FUNCTION_BLOCK "G310M_Code"
TITLE =G310M PLC1 TO EXCISTING DEGERMINATION SYSTEM
//COPYRIGHT:    (C) 2009  BUHLER AG, CH-9240 UZWIL, SWITZERLAND
//
//PRODUCT:      WinCoS_BIW01_09
//
//TITLE:        PLC1 TO EXCISTING DEGERMINATION SYSTEM
//                Machine group control
//                Maschinengruppensteuerung
//
//--------------------------------------------------------------------------------
//
//IDENT:        AUTHOR:             DEPT:                              DATE:
//
//P01_FB410.1.0 K.Renz              CSB41                              28.Jun.2010
//             1st Release
//
//--------------------------------------------------------------------------------
//
//PURPOSE:
//
//MANUAL :
//
//RESTRICTIONS:
//
//--------------------------------------------------------------------------------
AUTHOR : KR
FAMILY : USW
VERSION : 9.9


VAR
  Gr : "GCS7_GrpCtrlSub";	//Standard interface to group
  InOutValue1 : DINT ;	//Data for user
  InOutValue2 : DINT ;	//Data for user
  OutWayConflict : BOOL ;	//Data for user
  OutSelectionOk : BOOL ;	//Data for user
  CmdNewValue : BOOL ;	//Data for user
  CmdNewJob : BOOL ;	//Data for user
  OutCodeOK : BOOL ;	//Data for user
  InEndOfJob : BOOL ;	//Data for user
  staWayOk : BOOL ;	//Data for user
  EdgeStartRelease : BOOL ;	//Data for user
  USW8 : BOOL ;	//Data for user
  USW9 : BOOL ;	//Data for user
  USW10 : BOOL ;	//Data for user
  USW11 : BOOL ;	//Data for user
  USW12 : BOOL ;	//Data for user
  USW13 : BOOL ;	//Data for user
  USW14 : BOOL ;	//Data for user
  USW15 : BOOL ;	//Data for user
  A_3956_KCL01 : "GCS7_E_DigInput";	// DigInpCont
END_VAR
VAR_TEMP
  tmpEnable : BOOL ;
  tmpFlag : BOOL ;
  tmpCmdNext : BOOL ;
  tmpLocal : BOOL ;
  tmpAspOk : BOOL ;
  tmpHWStop : BOOL ;
  tmpInstanzDBNo : INT ;
END_VAR
BEGIN
NETWORK
TITLE =



NETWORK
TITLE =Read command from group control
//Parameter
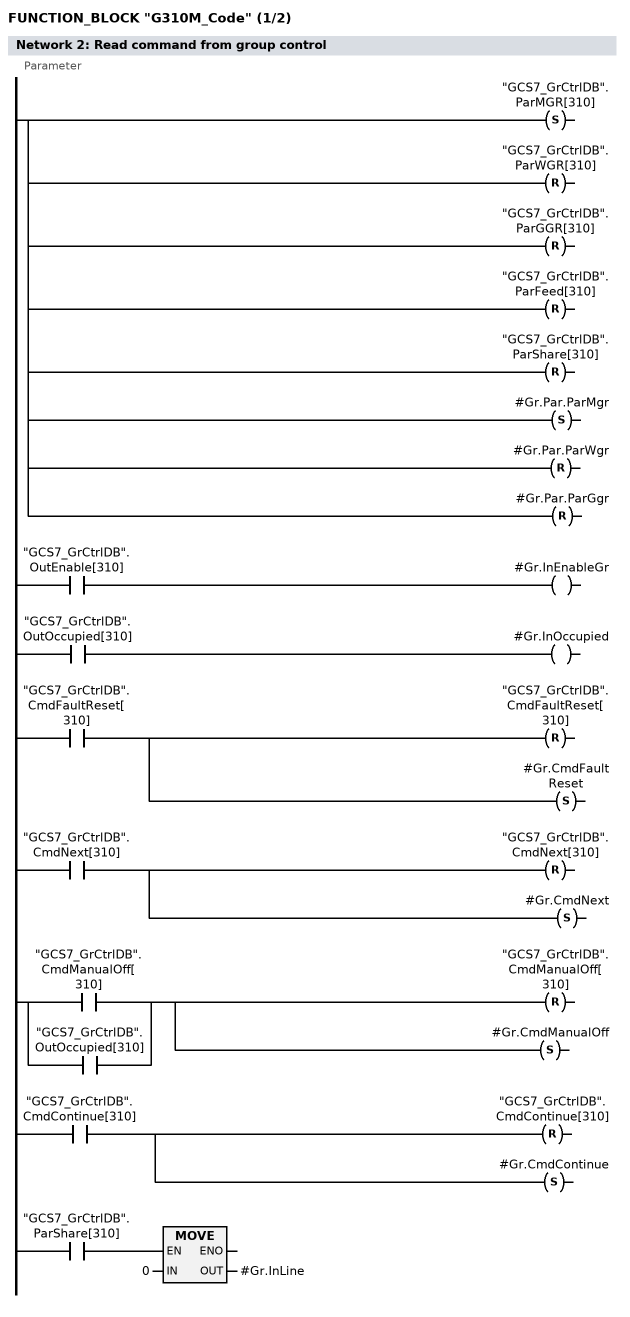
      SET   ;
      S     "GCS7_GrCtrlDB".ParMGR[310];
      R     "GCS7_GrCtrlDB".ParWGR[310];
      R     "GCS7_GrCtrlDB".ParGGR[310];
      R     "GCS7_GrCtrlDB".ParFeed[310];
      R     "GCS7_GrCtrlDB".ParShare[310];
      S     #Gr.Par.ParMgr;
      R     #Gr.Par.ParWgr;
      R     #Gr.Par.ParGgr;
//Command
      U     "GCS7_GrCtrlDB".OutEnable[310];
      =     #Gr.InEnableGr;
      U     "GCS7_GrCtrlDB".OutOccupied[310];
      =     #Gr.InOccupied;
      U     "GCS7_GrCtrlDB".CmdFaultReset[310];
      R     "GCS7_GrCtrlDB".CmdFaultReset[310];
      S     #Gr.CmdFaultReset;
      U     "GCS7_GrCtrlDB".CmdNext[310];
      R     "GCS7_GrCtrlDB".CmdNext[310];
      S     #Gr.CmdNext;
      U     "GCS7_GrCtrlDB".CmdManualOff[310];
      O     "GCS7_GrCtrlDB".OutOccupied[310];
      R     "GCS7_GrCtrlDB".CmdManualOff[310];
      S     #Gr.CmdManualOff;
      U     "GCS7_GrCtrlDB".CmdContinue[310];
      R     "GCS7_GrCtrlDB".CmdContinue[310];
      S     #Gr.CmdContinue;
//Init Line Number
      U     "GCS7_GrCtrlDB".ParShare[310];
      SPBN  WE00;
      L     0;
      T     #Gr.InLine;
WE00: NOP   0;
NETWORK
TITLE =Call Methode Control
// 1. Handle Interface PCControl
// 2. Prepare mode --> ModePassive,ModeActive,ModeIdling
// 3. Reset global flags of the group
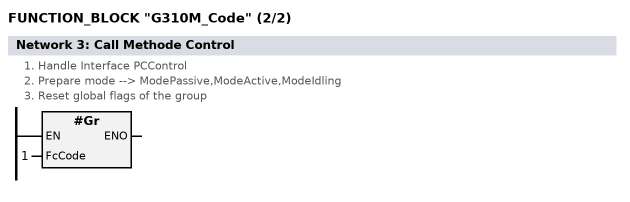
      CALL #Gr (
           FcCode                   := 1);
NETWORK
TITLE =Restart Idling Time

      L     #Gr.Par.ParIdling;
      L     2;
      >=I   ;
      SPB   IdTm;
      T     #Gr.Par.ParIdling;
IdTm: NOP   0;
      CLR   ;
      S     #Gr.CmdRestartIdling;
NETWORK
TITLE =Prepare global flags



NETWORK
TITLE =Set Pattern (Target position)



NETWORK
TITLE =Interlocking WayOk



NETWORK
TITLE =Interlocking Autostart

      CLR   ;
      R     #Gr.OutAutostart;
NETWORK
TITLE =Interlocking Enable
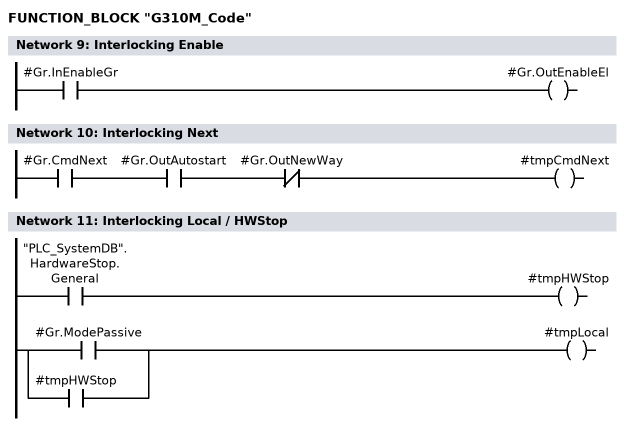

      U     #Gr.InEnableGr;
      =     #Gr.OutEnableEl;

NETWORK
TITLE =Interlocking Next

      U     #Gr.CmdNext;
      U     #Gr.OutAutostart;
      UN    #Gr.OutNewWay;
      =     #tmpCmdNext;

NETWORK
TITLE =Interlocking Local / HWStop

      U     "PLC_SystemDB".HardwareStop.General;
      =     #tmpHWStop;

      U     #Gr.ModePassive;
      O     #tmpHWStop;
      =     #tmpLocal;

NETWORK
TITLE =Interlocking Start Warning

      NOP   0;
//- Restart after fault --
      U     #Gr.CmdFaultReset;
      U     #Gr.VarFault;
      S     "SYS_StartWarningDB".Area[12].CmdResetStartWarning;
//- Run Timer --
      AUF   "G310M";
      CALL "GCS7_StartWarning" , "SYS_StartWarningDB" (
           InModeHigher             := FALSE,
           InArea                   := 12,
           InEnable                 := #Gr.OutEnableEl,
           InLocal                  := #tmpLocal,
           InStarted                := #Gr.VarStarted,
           InCmdNext                := #tmpCmdNext,
           OutCmdNext               := #tmpCmdNext,
           OutStartwarning          := #Gr.VarStartwarning);
//- Store Startwarning done  --
//- Reset Autostart --
      U     "SYS_StartWarningDB".TmpArea.OutStartReleaseRunningL;
      FN    #EdgeStartRelease;
      U     #Gr.VarFault;
      R     #Gr.OutAutostart;
NETWORK
TITLE ==A-3956-KCL01 : EXCISTING DEGERMINATING SYSTEM

      NOP   0;
//-InLocal---
      U     #tmpLocal;
      =     #A_3956_KCL01.InLocal;
//
//-Monitoring---
      CLR   ;
      =     #A_3956_KCL01.InMonTrue;
      CLR   ;
      =     #A_3956_KCL01.InMonFalse;
//
//-PreAlarm---
      CLR   ;
      =     #A_3956_KCL01.InPreAlarmTrue;
      CLR   ;
      =     #A_3956_KCL01.InPreAlarmFalse;
//
//-Additional commands---
//      CLR
//      S     #A_3956_KCL01.CmdRunTimeOutTime
//
//-Read inputs---
      U     "A_3956_KCL01_I1";
      =     #A_3956_KCL01.InpTrue;
      U     "PLC_SystemDB".GlobalFlags.UnloadingKilning;
      =     #A_3956_KCL01.InHWStop;
      U     "PLC_DPInfo".Master[1].SlavesError[115];
      =     #A_3956_KCL01.InDPFault;
//
//-Set Parameters---
//
//-Call object control---
      CALL #A_3956_KCL01 ;
//
//-Write outputs---
NETWORK
TITLE =Test Fault

      U     #A_3956_KCL01.StFault;
      =     #Gr.VarFault;
NETWORK
TITLE =Test Warning

      CLR   ;
      =     #Gr.OutWarning;
NETWORK
TITLE =Test Stopped
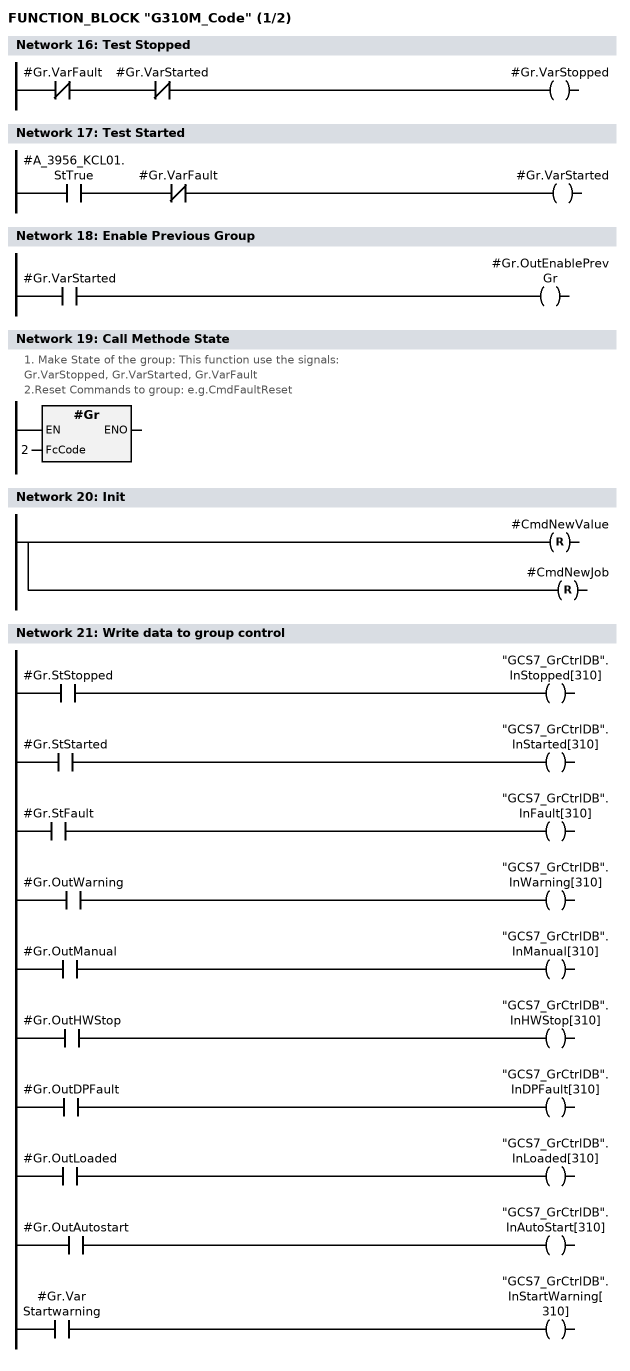

      UN    #Gr.VarFault;
      UN    #Gr.VarStarted;
      =     #Gr.VarStopped;
NETWORK
TITLE =Test Started

//      UN    #Gr.VarStopped
      U     #A_3956_KCL01.StTrue;
      UN    #Gr.VarFault;
      =     #Gr.VarStarted;
NETWORK
TITLE =Enable Previous Group

      U     #Gr.VarStarted;
      =     #Gr.OutEnablePrevGr;
NETWORK
TITLE =Call Methode State
//1. Make State of the group: This function use the signals:
//        Gr.VarStopped, Gr.VarStarted, Gr.VarFault
//2.Reset Commands to group: e.g.CmdFaultReset
      CALL #Gr (
           FcCode                   := 2);
NETWORK
TITLE =Init

      SET   ;
      R     #CmdNewValue;
      R     #CmdNewJob;
NETWORK
TITLE =Write data to group control

      U     #Gr.StStopped;
      =     "GCS7_GrCtrlDB".InStopped[310];
      U     #Gr.StStarted;
      =     "GCS7_GrCtrlDB".InStarted[310];
      U     #Gr.StFault;
      =     "GCS7_GrCtrlDB".InFault[310];
      U     #Gr.OutWarning;
      =     "GCS7_GrCtrlDB".InWarning[310];
      U     #Gr.OutManual;
      =     "GCS7_GrCtrlDB".InManual[310];
      U     #Gr.OutHWStop;
      =     "GCS7_GrCtrlDB".InHWStop[310];
      U     #Gr.OutDPFault;
      =     "GCS7_GrCtrlDB".InDPFault[310];
      U     #Gr.OutLoaded;
      =     "GCS7_GrCtrlDB".InLoaded[310];
      U     #Gr.OutAutostart;
      =     "GCS7_GrCtrlDB".InAutoStart[310];
      U     #Gr.VarStartwarning;
      =     "GCS7_GrCtrlDB".InStartWarning[310];
NETWORK
TITLE =End of block
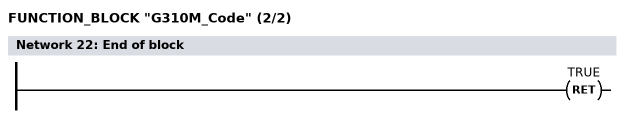

      BE    ;

END_FUNCTION_BLOCK

